// Converts TcLog.LogLevels into Tc2_System.AdsLog_MsgType.
//{attribute 'hide'}
FUNCTION INTERNAL LogLevelToAdsLogMsgType : DWORD
VAR_INPUT
  level : LogLevel;
END_VAR

CASE level OF
	LogLevel.Debug,
	LogLevel.Information:
		LogLevelToAdsLogMsgType := Tc2_System.AdsLog_MsgType_Hint;
		
	LogLevel.Warning:
		LogLevelToAdsLogMsgType := Tc2_System.AdsLog_MsgType_Warn;
		
	LogLevel.Error,
	LogLevel.Fatal:
		LogLevelToAdsLogMsgType := Tc2_System.AdsLog_MsgType_Error;
ELSE
	LogLevelToAdsLogMsgType := Tc2_System.AdsLog_MsgType_Hint;
END_CASE

END_FUNCTION

(* stored: Version 1.1.0.1
   POU LogLevelToAdsLogMsgType: Id {0deed475-5a07-4f2a-a95a-4191ee389a8c}, SpecialFunc None *)
